TYPE E_TestPhase :
(
    TEST_IDLE       := 0,
    TEST_SETUP      := 1,
    TEST_EXECUTE    := 2,
    TEST_SETTLE     := 3,
    TEST_VERIFY     := 4,
    TEST_TEARDOWN   := 5,
    TEST_DONE       := 6
);
END_TYPE

(* stored: Version 1.1.0.1
   DUT E_TestPhase: Id {7418DA1F-F211-1098-245A-D675C0F76947} *)
